% RSLogix 500 project AB_PROJECT1_V1_0_pump_control.RSS, saved by version 8.30.00.16 %
PROJECT "AB"    % processor: Bul.1763 MicroLogix 1100 Series A %

PROGRAM FILES
  LAD 2   5 rungs
  LAD 3, 4, 5, 6, 7, 8, 9, 10, 11, 12, 13, 14, 15, 16: only END

DATA FILES
  O0 OUTPUT  4 elements
  I1 INPUT  6 elements
  S2 STATUS  66 elements
  B3 BINARY  32 elements
  T4 TIMER  40 elements
  C5 COUNTER  32 elements
  R6 CONTROL  16 elements
  N7 INTEGER  105 elements
  F8 FLOAT  1 elements

LADDER 2
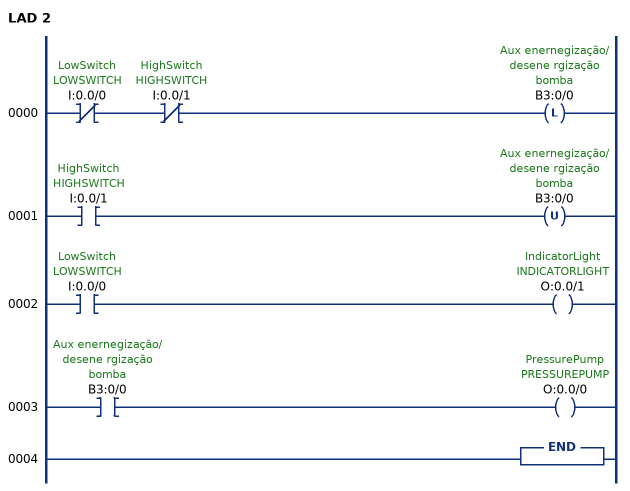
% Rung: 0 %
SOR XIO I:0.0/0 XIO I:0.0/1 OTL B3:0/0 EOR
%   I:0.0/0  LOWSWITCH  "LowSwitch" %
%   I:0.0/1  HIGHSWITCH  "HighSwitch" %
%   B3:0/0  "Aux enernegização/desene rgização bomba" %
% Rung: 1 %
SOR XIC I:0.0/1 OTU B3:0/0 EOR
%   I:0.0/1  HIGHSWITCH  "HighSwitch" %
%   B3:0/0  "Aux enernegização/desene rgização bomba" %
% Rung: 2 %
SOR XIC I:0.0/0 OTE O:0.0/1 EOR
%   I:0.0/0  LOWSWITCH  "LowSwitch" %
%   O:0.0/1  INDICATORLIGHT  "IndicatorLight" %
% Rung: 3 %
SOR XIC B3:0/0 OTE O:0.0/0 EOR
%   B3:0/0  "Aux enernegização/desene rgização bomba" %
%   O:0.0/0  PRESSUREPUMP  "PressurePump" %
% Rung: 4 %
SOR END EOR

DATA TABLE (non-zero values as saved)
DATA B3
% B3:0 % 0X0001 0X0000 0X0000 0X0000 0X0000 0X0000 0X0000 0X0000 0X0000 0X0000
